FUNCTION_BLOCK POUPOU
VAR_INPUT
END_VAR
VAR_OUTPUT
END_VAR
VAR
END_VAR

END_FUNCTION_BLOCK

(* stored: Version 1.1.0.1, ProductVersion 3.1.4024.9
   POU POUPOU: Id {995a384b-0e51-4c7e-aa8e-9ba6c0096ea3}, SpecialFunc None *)
